TYPE Sub_Step :
STRUCT
	Step	: INT;
	
	bBuzy	: BOOL;
	bDone	: BOOL;
	bError	: BOOL;
END_STRUCT
END_TYPE

(* stored: Version 1.1.0.1, ProductVersion 3.1.4026.13
   DUT Sub_Step: Id {314ddef8-b01a-495a-b492-e48a9887e90b} *)
